// TIA Portal V20 export
// export: Created 2025-12-01T14:57:04.0292888Z, ExportSetting None, DisplayName Totally Integrated Automation Portal, DisplayVersion V20 Update 3, DisplayName TIA Portal Openness, DisplayVersion V20 Update 3, DisplayName TIA Portal Version Control Interface, DisplayVersion V20 Update 3, DisplayName STEP 7 Professional, DisplayVersion V20 Update 3, DisplayName STEP 7 Safety, DisplayVersion V20 Update 2, DisplayName WinCC Basic/Comfort/Advanced, DisplayVersion V20 Update 3, DisplayName WinCC Professional, DisplayVersion V20 Update 3, DisplayName WinCC Unified, DisplayVersion V20 Update 3
FUNCTION "FC703_JDT02EmiJdTMensaje" : Void   // FC703, LAD
TITLE = "EmiJdTMensaje" - Emision de Mensajes
{ S7_Optimized_Access := 'FALSE' }
AUTHOR : TRACKING
NAME : 20141014
VERSION : 4.0
// - Inicializaciones
// - Distrubucion
// - Recoger el Mensaje ACKN
// - Recoger el Mensaje PING o Lista de Eventos
// - Emision del Mensaje
// stored: AutoNumber false, SetENOAutomatically false
   VAR_TEMP
      DBEmiJdT : Word;   // Num. DB de Emision al JdT
      DBUltimoEmi : Word;   // Num. DB del Ultimo Mensaje a Emitir
      DBEmiAK : Word;   // Num. DB del Mensaje AK a Emitir
      Longitud : UDInt;   // Longitud del Mensaje
      CantidadBytes : UDInt;   // Cantidad de Bytes del Mensaje a Enviar
      ReturnValor : Int;   // Temporal
      POrigen : Any;   // Puntero para transferencias y emision
      PDestino : Any;   // Puntero para transferencias
   END_VAR
BEGIN

NETWORK
TITLE = Inicializaciones
// - Inicializa las variables de los DB's
// - Comprueba que el enlace esta activo "EnlaceCP_OK"
// -------------------------------------------------------------------------------------------
// Si trabaja sin Agencia  2018 01 24
      SET;
      AN    "Activar_JDT02";  // Mirar si se trabaja con agencia
      JC    Final;

// ------------------------------------------------------------------------------------------
// Inicializa las variables de los DB's

      L     "JDT2_NDB_EmiMensaje";  // Cogemos el Numero del DB de EmisionMensaje
      T     #DBEmiJdT;
      L     "JDT2_NDB_UltimoEmi";  // Cogemos el Numero del DB de UltimaEmision
      T     #DBUltimoEmi;
      L     "JDT2_NDB_AKEmi";  // Cogemos el Numero del DB de EmisionAK
      T     #DBEmiAK;

// ------------------------------------------------------------------------------------------
// Comprueba el Enlace esta correcto

      A     "DB701_JDT02StatusCOM".EnlaceCP_OK;  // Mirar Si esta el EnlaceCP Activo
      JC    ExisteConexion;  // El EnlaceCP esta OK

// Reseteamos las variables porque El enlaceCP NOK

      R     "DB891_VariablesTCP".TSEND_JdT_PLC_Req_JDT02;  // Resetear Variables
      R     "DB891_VariablesTCP".TSEND_JdT_PLC_Done_JDT02;
      R     "DB891_VariablesTCP".TSEND_JdT_PLC_Error_JDT02;
      R     "DB891_VariablesTCP".TSEND_JdT_PLC_Busy_JDT02;


      JU    Final;  // Finalizar


NETWORK
TITLE = Distribución
// Hay que seguir este orden:
// - Hay que emitir mensaje
// - Hay que recoger el mensaje ACKN
// - Hay que recoger el mensaje PING o Lista de Eventos
ExisteConexion:NOP   0;

// ------------------------------------------------------------------------------------------
// Hay que emitir mensaje

      L     0;  // Ya tenemos mensaje a Emitir
      LAR1;
      OPN   DB [#DBEmiJdT];
      L     DBB [AR1, P#0.0];
      L     0;
      <>I;
      JC    EmitirMensaje;  // Ir a Emitir

// ------------------------------------------------------------------------------------------
// Hay que recoger Mensaje ACKN para emitir

      L     0;
      LAR1;
      OPN   DB [#DBEmiAK];
      L     DBB [AR1, P#0.0];
      L     2;
      ==I;
      JC    EmitirEvento_AcuseRecibo;  // Ir a Recoger el mensaje AK

// ------------------------------------------------------------------------------------------
// Hay que recoger Mensaje PING o Lista de Eventos para Emitir

      L     0;
      LAR1;
      OPN   DB [#DBUltimoEmi];
      L     DBB [AR1, P#0.0];
      L     2;
      ==I;
      JC    EmitirEvento;  // Ir a Recoger el mensaje KA o de Eventos

      JU    Final;



NETWORK
TITLE = Recoger el Mensaje ACKN - Confirmacion
// Pasos a Seguir:
// - Calcular la Longitud del Mensaje (Puede ser variable)
// - Generamos los punteros Origen y Destino
// - Transferir el Mensaje para Emitir
// - Borrar el Mensaje AK, para decir que lo hemos tratado, y Resetear Variables
// - Emitimos el Mensaje
EmitirEvento_AcuseRecibo:NOP   0;

// ------------------------------------------------------------------------------------------
// 1º Paso - Calcular la longitud del Mensaje

      CALL  "FC890_EtiqChar_EtiqDInt"
      ( DB_String   := "JDT2_NDB_AKEmi",
        Long_String := 5,
        Offset_Ini  := 20,
        Valor       := #Longitud
      );

      L     #Longitud;
      T     #CantidadBytes;

// ------------------------------------------------------------------------------------------
// 2º Paso - Generamos los punteros Origen y Destino

      CALL  "FC897_Generar_PointerAny"
      ( TYP           := 16#10,
        DataTyp       := 16#02,
        repeatcounter := #CantidadBytes,  // Tamaño del mensaje
        DB_Number     := "JDT2_NDB_AKEmi",  // DB donde esta guardado el EmisionAK
        storearea     := 16#84,
        storeaddresse := 16#0000_0000,
        Any_Pointer   := #POrigen  // Puntero del EmisionAK
      );

      CALL  "FC897_Generar_PointerAny"
      ( TYP           := 16#10,
        DataTyp       := 16#02,
        repeatcounter := #CantidadBytes,  // Tamaño del mensaje
        DB_Number     := "JDT2_NDB_EmiMensaje",  // DB donde guardar el EmisionMensaje
        storearea     := 16#84,
        storeaddresse := 16#0000_0000,
        Any_Pointer   := #PDestino  // Puntero del Mensaje a Enviar
      );

// ------------------------------------------------------------------------------------------
// 3º Paso - Transferir en Mensaje para emitir

      CALL  BLKMOV
      ( SRCBLK  := #POrigen,
        RET_VAL := #ReturnValor,
        DSTBLK  := #PDestino
      );

// ------------------------------------------------------------------------------------------
// 4º Paso - Borrar el Mensaje AK y Resetear variables internas

      CALL  "FC898_BorrarMensaje"
      ( DB_A_RESET := "DB706_JDT02EmisionAK"  // ¿Hay que borrar asi?
      );  // Damos por acabado el envio del mensaje

      SET;  // Ya hay Actividad
      R     "DB701_JDT02StatusCOM".SinActividad;

// ------------------------------------------------------------------------------------------
// 5º Paso - Pasamos a Emitir el Mensaje

      L     #CantidadBytes;
      T     "DB701_JDT02StatusCOM".EmiJdT_Longitud;  // Guardamos la longitud para la Emision
      JU    EmitirMensaje;



NETWORK
TITLE = Recoger el Mensaje KA o Lista de Eventos
// Pasos a Seguir:
// - Calcular la Longitud del Mensaje(Puede ser variable)
// - Generamos los punteros Origen y Destino
// - Transferir el Mensaje para Emitir
// - Borrar el Mensaje AK, para decir que lo hemos tratado, y Resetear Variables
// - Emitimos el Mensaje
EmitirEvento:NOP   0;

// ------------------------------------------------------------------------------------------
// 1º Paso - Calcular la longitud del Mensaje

      CALL  "FC890_EtiqChar_EtiqDInt"
      ( DB_String   := "JDT2_NDB_UltimoEmi",
        Long_String := 5,
        Offset_Ini  := 20,
        Valor       := #Longitud
      );

      L     #Longitud;
      T     #CantidadBytes;

// ------------------------------------------------------------------------------------------
// 2º Paso - Generamos los punteros Origen y Destino

      CALL  "FC897_Generar_PointerAny"
      ( TYP           := 16#10,
        DataTyp       := 16#02,
        repeatcounter := #CantidadBytes,  // Tamaño del mensaje
        DB_Number     := "JDT2_NDB_UltimoEmi",  // DB donde esta guardado el UltimoMensaje
        storearea     := 16#84,
        storeaddresse := 16#0000_0000,
        Any_Pointer   := #POrigen  // Puntero del UltimoMensaje
      );

      CALL  "FC897_Generar_PointerAny"
      ( TYP           := 16#10,
        DataTyp       := 16#02,
        repeatcounter := #CantidadBytes,  // Tamaño del mensaje
        DB_Number     := "JDT2_NDB_EmiMensaje",  // DB donde guardar el Emisio del Mensaje
        storearea     := 16#84,
        storeaddresse := 16#0000_0000,
        Any_Pointer   := #PDestino  // Puntero del Mensaje a Enviar
      );

// ------------------------------------------------------------------------------------------
// 3º Paso - Transferir

      CALL  BLKMOV
      ( SRCBLK  := #POrigen,
        RET_VAL := #ReturnValor,
        DSTBLK  := #PDestino
      );

// ------------------------------------------------------------------------------------------
// 4º Paso - Borrar el Mensaje Tratado y Resetear variables internas

      SET;  // Ya hay Actividad
      R     "DB701_JDT02StatusCOM".SinActividad;

// Parar Borrar el Mensaje hay que saber de que tipo es:
// KA o Lista de Eventos - Porque se hace cosas diferentes

      L     0;
      LAR1;
      OPN   DB [#DBUltimoEmi];
      L     DBD [AR1, P#24.0];
      L     'PING';
      <>I;
      JC    _040;  // Si no es KA hay que borrarlo entero

// Es Mensaje KA - Borrar todo el Mensaje
      CALL  "FC898_BorrarMensaje"
      ( DB_A_RESET := "DB705_JDT02UltimoEnviado"  // ¿Hay que borrar asi?
      );  // Damos por acabado el envio del mensaje KA

      JU    _041;

// Es Mnesaje de Lista de Eventos lo damos por tratado
_040: OPN   DB [#DBUltimoEmi];  // Damos por enviado el mensaje de Evento
      L     'N';
      T     DBB [AR1, P#0.0];

      JU    _041;

// ------------------------------------------------------------------------------------------
// 5º Paso - Pasamos a Emitir el Mensaje

_041: L     #CantidadBytes;
      T     "DB701_JDT02StatusCOM".EmiJdT_Longitud;  // Guardamos la longitud para la Emision
      JU    EmitirMensaje;



NETWORK
TITLE = Emision del Mensaje
// Pasos a Seguir
// - Control de la Emision
// - Calcular el puntero de lo que tenemos que emitir
// - Emision del Mensaje
// - Comprobacion del Mensaje Enviado
EmitirMensaje:NOP   0;

// ------------------------------------------------------------------------------------------
// 1º Paso - Control de la Emision

      AN    "DB891_VariablesTCP".TSEND_JdT_PLC_Busy_JDT02;
      AN    "DB891_VariablesTCP".TSEND_JdT_PLC_Req_JDT02;
      AN    "DB891_VariablesTCP".TSEND_JdT_PLC_Flanco_JDT02;
      =     "DB891_VariablesTCP".TSEND_JdT_PLC_Flanco_JDT02;

      A     "DB891_VariablesTCP".TSEND_JdT_PLC_Flanco_JDT02;
      AN    "DB891_VariablesTCP".TSEND_JdT_PLC_Req_JDT02;
      S     "DB891_VariablesTCP".TSEND_JdT_PLC_Req_JDT02;


// ------------------------------------------------------------------------------------------
// 2º Paso - Generar el Puntero de lo que se tiene que Emitir

      CALL  "FC897_Generar_PointerAny"
      ( TYP           := 16#10,
        DataTyp       := 16#02,
        repeatcounter := "DB701_JDT02StatusCOM".EmiJdT_Longitud,  // Tamaño del mensaje
        DB_Number     := "JDT2_NDB_EmiMensaje",  // DB donde esta guardado el EmisionMensaje
        storearea     := 16#84,
        storeaddresse := 16#0000_0000,
        Any_Pointer   := #POrigen  // Puntero del EmisionMensaje
      );

// ------------------------------------------------------------------------------------------
// 2º Paso - Emision del Mensaje

      CALL  TSEND, "DB898_TSEND_JdT_PLC_JDT02"
      ( REQ    := "DB891_VariablesTCP".TSEND_JdT_PLC_Flanco_JDT02,
        ID     := W#16#3,
        LEN    := "DB701_JDT02StatusCOM".EmiJdT_Longitud,
        DONE   := "DB891_VariablesTCP".TSEND_JdT_PLC_Done_JDT02,
        BUSY   := "DB891_VariablesTCP".TSEND_JdT_PLC_Busy_JDT02,
        ERROR  := "DB891_VariablesTCP".TSEND_JdT_PLC_Error_JDT02,
        STATUS := "DB891_VariablesTCP".TSEND_JdT_PLC_Status_JDT02,
        DATA   := #POrigen
      );



// ------------------------------------------------------------------------------------------
// 3º Paso - Comprobacion del Mensaje Enviado

      A     "DB891_VariablesTCP".TSEND_JdT_PLC_Req_JDT02;  // Si llega Error en la Emision
      AN    "DB891_VariablesTCP".TSEND_JdT_PLC_Done_JDT02;  // Restear
      A     "DB891_VariablesTCP".TSEND_JdT_PLC_Error_JDT02;
      S     "DB701_JDT02StatusCOM".EmiJdT_Reset;
      R     "DB891_VariablesTCP".TSEND_JdT_PLC_Req_JDT02;

      A     "DB891_VariablesTCP".TSEND_JdT_PLC_Req_JDT02;  // Si llega que la Emision es OK
      A     "DB891_VariablesTCP".TSEND_JdT_PLC_Done_JDT02;
      AN    "DB891_VariablesTCP".TSEND_JdT_PLC_Error_JDT02;
      R     "DB891_VariablesTCP".TSEND_JdT_PLC_Req_JDT02;

      JCN   NoEmitidoMensaje;

      R     "DB701_JDT02StatusCOM".EmiJdT_PeticionActiva;
      CALL  "FC898_BorrarMensaje"
      ( DB_A_RESET := "DB703_JDT02EmisionMensaje"  // ¿Hay que borralo asi?
      );

NoEmitidoMensaje:JU    Final;


NETWORK
TITLE = Finalizar
// - Finaliza la función
Final:NOP   0;

END_FUNCTION
